(* IEC 61131-3 sources: AXOpen/src/components.pneumatics/ctrl/src, 1 file *)

(* ---- AxoCylinder.st ---- *)
USING AXOpen.Core;
USING AXOpen.Messaging;
USING AXOpen.Messaging.Static;

NAMESPACE AXOpen.Components.Pneumatics
    {S7.extern=ReadWrite}
    CLASS AxoCylinder EXTENDS AXOpen.Core.AxoComponent
        VAR PUBLIC
            {#ix-attr:[Container(Layout.Wrap)]}
            {#ix-attr:[ComponentHeader()]}
            {#ix-set:AttributeName = "<#Move to work#>"}
            _MoveToWorkTask : AxoTask;

            {#ix-attr:[ComponentHeader()]}
            {#ix-set:AttributeName = "<#Move to home#>"}
            _MoveToHomeTask : AxoTask;

            {#ix-attr:[ComponentDetails("Tasks")]}
            {#ix-set:AttributeName = "<#Stop#>"}
            _StopTask : AxoTask;

            {#ix-attr:[Container(Layout.Stack)]}
            {#ix-attr:[ComponentDetails("Signals")]}
            {#ix-attr:[ReadOnly()]}
            {#ix-set:AttributeName = "<#Home sensor#>"}
            _HomeSensor : BOOL;

            {#ix-attr:[ComponentDetails("Signals")]}
            {#ix-attr:[ReadOnly()]}
            {#ix-set:AttributeName = "<#Work sensor#>"}
            _WorkSensor : BOOL;

            {#ix-attr:[Container(Layout.Stack)]}
            {#ix-attr:[ComponentDetails("Signals")]}
            {#ix-attr:[ReadOnly()]}
            {#ix-set:AttributeName = "<#Move home signal#>"}
            _MoveHomeSignal : BOOL;

            {#ix-attr:[ComponentDetails("Signals")]}
            {#ix-attr:[ReadOnly()]}
            {#ix-set:AttributeName = "<#Move work signal#>"}
            _MoveWorkSignal : BOOL;

            _Messenger : AXOpen.Messaging.Static.AxoMessenger;
        END_VAR

        VAR PRIVATE
            _MoveToWorkIsSuspended : BOOL;
            _MoveToHomeIsSuspended : BOOL;

            _MoveToWorkIsBusy : BOOL;
            _MoveToHomeIsBusy : BOOL;

            _context : IAxoContext;
        END_VAR

        ///<summary>
        /// Runs tasks and logic of this component.
        /// >[!IMPORTANT] This method or one of its overloads must be called cyclically.
        ///</summary>
        METHOD PUBLIC Run
            VAR_INPUT
                parent : IAxoObject;
                homeSensor : BOOL;
                workSensor : BOOL;
            END_VAR
            VAR_OUTPUT
                moveHomeSignal : BOOL;
                moveWorkSignal : BOOL;
            END_VAR

            IF (parent = NULL) THEN
                RETURN;
            END_IF;

            IF _context = NULL THEN
                SUPER.Run(parent);
                _context := THIS.GetContext();
            END_IF;

            SUPER.Run(parent);

            _Messenger.Serve(THIS);

            _Messenger.ActivateOnCondition(UINT#3, workSensor AND homeSensor, eAxoMessageCategory#Error);

            IF(_StopTask.Execute(THIS)) THEN
                moveHomeSignal := FALSE;
                moveWorkSignal := FALSE;
                _MoveToHomeTask.Restore();
                _MoveToWorkTask.Restore();
                _StopTask.DoneWhen(TRUE);
            END_IF;

            IF(_MoveToWorkTask.Execute(THIS)) THEN
                moveHomeSignal := FALSE;
                moveWorkSignal := TRUE;
                _MoveToWorkTask.DoneWhen(workSensor);
                _MoveToHomeTask.Restore();
            END_IF;

            _MoveToWorkIsBusy := _MoveToWorkTask.IsBusy();

           _Messenger.ActivateOnCondition(UINT#1, (_MoveToWorkIsBusy AND NOT _MoveToWorkIsSuspended AND _MoveToWorkTask.Duration >= T#10S), eAxoMessageCategory#Error);
           _Messenger.ActivateOnCondition(UINT#9, (_MoveToWorkTask.IsDone() AND NOT workSensor), eAxoMessageCategory#Warning);

            IF(_MoveToHomeTask.Execute(THIS)) THEN
                moveHomeSignal := TRUE;
                moveWorkSignal := FALSE;
                _MoveToHomeTask.DoneWhen(homeSensor);
                _MoveToWorkTask.Restore();
            END_IF;

            _MoveToHomeIsBusy := _MoveToHomeTask.IsBusy();

            _Messenger.ActivateOnCondition(UINT#2, (_MoveToHomeIsBusy AND NOT _MoveToHomeIsSuspended AND _MoveToHomeTask.Duration >= T#10S), eAxoMessageCategory#Error);
            _Messenger.ActivateOnCondition(UINT#8, (_MoveToHomeTask.IsDone() AND NOT homeSensor), eAxoMessageCategory#Warning);

            IF _MoveToWorkIsSuspended THEN
                moveWorkSignal := FALSE;
            END_IF;

            _Messenger.ActivateOnCondition(UINT#4, _MoveToWorkIsSuspended AND _MoveToWorkIsBusy, eAxoMessageCategory#Info);

            IF _MoveToHomeIsSuspended THEN
                moveHomeSignal := FALSE;
            END_IF;

           _Messenger.ActivateOnCondition(UINT#5, _MoveToHomeIsSuspended AND _MoveToHomeIsBusy, eAxoMessageCategory#Info);

            _HomeSensor := homeSensor;
            _WorkSensor := workSensor;

            _MoveHomeSignal := moveHomeSignal;
            _MoveWorkSignal := moveWorkSignal;

        END_METHOD

        METHOD PROTECTED OVERRIDE ManualControl
            THIS._isManuallyControllable := true;
        END_METHOD

        ///<summary>
        /// Restores this component into intial state.
        ///</summary>
        METHOD PUBLIC OVERRIDE Restore
            _MoveToWorkTask.Restore();
            _MoveToHomeTask.Restore();
            _StopTask.Restore();
        END_METHOD

        ///<summary>
		/// Invokes the movement to the work position and returns the task state.
        ///</summary>
        METHOD PUBLIC MoveToWork : IAxoTaskState
            MoveToWork := _MoveToWorkTask.Invoke(THIS);
        END_METHOD

        ///<summary>
		/// Invokes the movement to the home position and returns the task state.
        ///</summary>
        METHOD PUBLIC MoveToHome : IAxoTaskState
            MoveToHome := _MoveToHomeTask.Invoke(THIS);
        END_METHOD

        ///<summary>
		/// Stops any movement.
        ///</summary>
        METHOD PUBLIC Stop : IAxoTaskState
            Stop := _StopTask.Invoke(THIS);
        END_METHOD

        ///<summary>
        /// Suspends the movement to the work position while the condition is 'true'. Task remains still executing.
        ///</summary>
        METHOD PUBLIC SuspendMoveToWorkWhile
            VAR_INPUT
                Condition : BOOL;
            END_VAR

            IF(Condition) THEN
                _moveWorkSignal := FALSE;
            END_IF;
            _Messenger.ActivateOnCondition(UINT#4, Condition AND _MoveToWorkTask.IsBusy(), eAxoMessageCategory#Info);
            _MoveToWorkIsSuspended := Condition;
        END_METHOD

        ///<summary>
        /// Suspends the movement to the home position while the condition is 'true'. Task remains still executing.
        ///</summary>
        METHOD PUBLIC SuspendMoveToHomeWhile
            VAR_INPUT
                Condition : BOOL;
            END_VAR

            IF(Condition) THEN
                _moveHomeSignal := FALSE;
            END_IF;
            _Messenger.ActivateOnCondition(UINT#5, Condition AND _MoveToHomeTask.IsBusy(), eAxoMessageCategory#Info);
            _MoveToHomeIsSuspended := Condition;
        END_METHOD

        ///<summary>
        /// Aborts the movement to the work position when the condition is 'true' and restores the respective task.
        ///</summary>
        METHOD PUBLIC AbortMoveToWorkWhen
            VAR_INPUT
                Condition : BOOL;
            END_VAR

            IF(Condition) THEN
                _moveWorkSignal := FALSE;
                _MoveToWorkTask.Abort();
                _Messenger.Activate(UINT#6, eAxoMessageCategory#Info);
            END_IF;
            _MoveToWorkTask.SetIsDisabled(Condition);
        END_METHOD

        ///<summary>
        /// Aborts the movement to the home position when the condition is 'true' and restores the respective task.
        ///</summary>
        METHOD PUBLIC AbortMoveToHomeWhen
            VAR_INPUT
                Condition : BOOL;
            END_VAR

            IF(Condition) THEN
                _moveHomeSignal := FALSE;
                _Messenger.Activate(UINT#7, eAxoMessageCategory#Info);
                _MoveToHomeTask.Abort();
            END_IF;
            _MoveToHomeTask.SetIsDisabled(Condition);
        END_METHOD
    END_CLASS
END_NAMESPACE
